// TIA Portal V16 export
// export: Created 2022-11-17T15:49:21.0130666Z, ExportSetting WithDefaults, DisplayName Totally Integrated Automation Portal, DisplayVersion V16 Update 6, DisplayName TIA Portal Version Control Interface, DisplayVersion V16 Update 2, DisplayName TIA Portal Openness, DisplayVersion V16 Update 6, DisplayName SINAMICS Startdrive Advanced, DisplayVersion V16 Update 5, DisplayName SINAMICS Startdrive G130, G150, S120, S150, SINAMICS MV, S210, DisplayVersion V16 Update 5, DisplayName SINAMICS Startdrive G110M, G120, G120C, G120D, G120P, G115D, DisplayVersion V16 Update 5, DisplayName STEP 7 Professional, DisplayVersion V16 Update 6, DisplayName STEP 7 Safety, DisplayVersion V16, DisplayName WinCC Advanced, DisplayVersion V16 Update 6
FUNCTION "FC27_PosSelfcEncoder" : Void   // FC27, LAD
TITLE = Pallet positioning with selfcentering system and encoder
{ S7_Optimized_Access := 'FALSE' }
AUTHOR : Robopac
VERSION : 0.0
// stored: AutoNumber false, IsIECCheckEnabled false, SetENOAutomatically false, UDAEnableTagReadback false
   VAR_TEMP
      Ch7ValmmEnco1 : DInt;
      Ch7ValmmEnco2 : DInt;
      PalletLenghtdiv2 : Int;
      PosToReach : Int;
      PosToDecelation : Int;
      WTemp1 : Int;
      DWTemp1 : DInt;
      DWTemp2 : DInt;
   END_VAR
   VAR_TEMP   // added for the SCL form of the ladder/FBD networks
      _w1 : Bool;
      _w2 : Bool;
   END_VAR
BEGIN

REGION Network 1: Delay on pallet positioning left
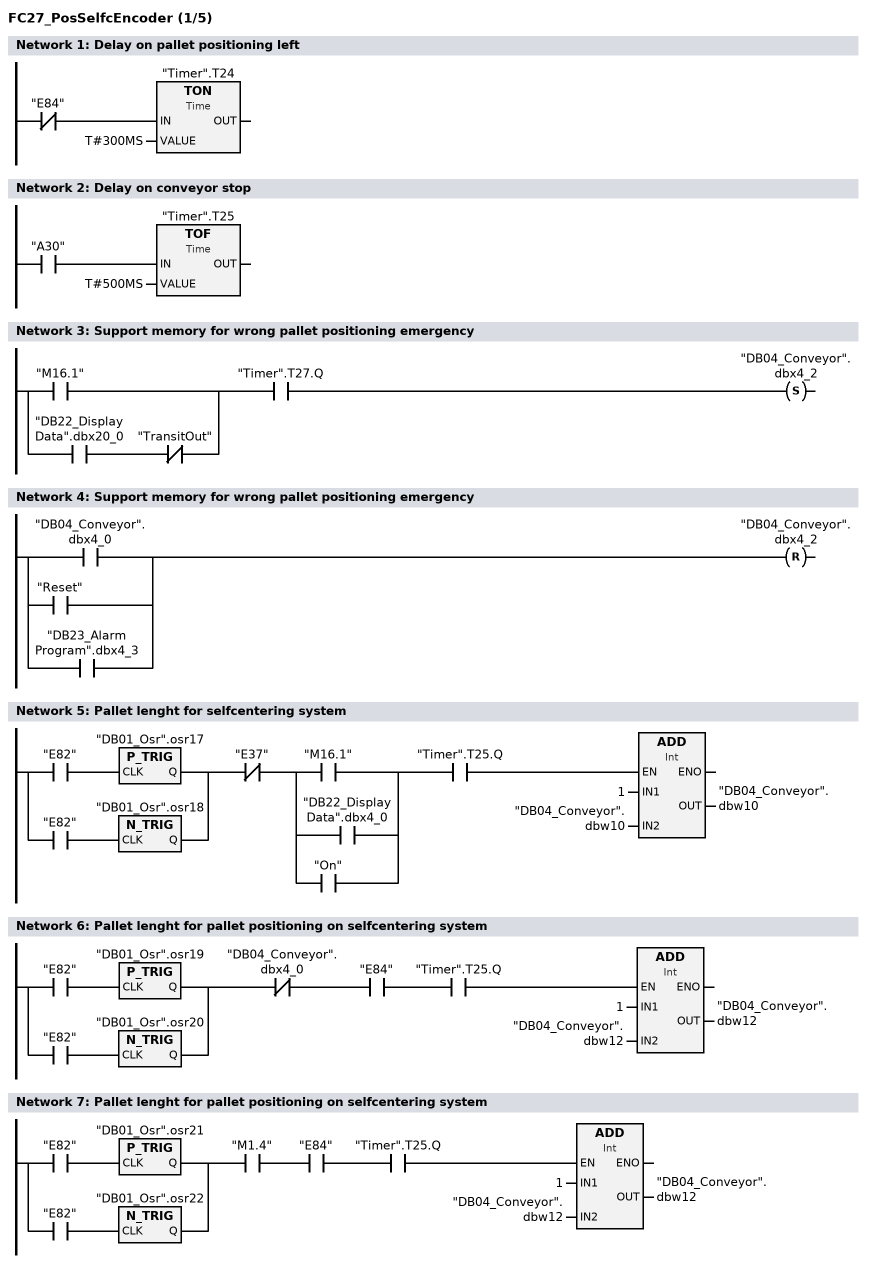
   "Timer".T24.TON(IN := NOT "E84", PT := T#300MS);   // TON coil
END_REGION

REGION Network 2: Delay on conveyor stop
   "Timer".T25.TOF(IN := "A30", PT := T#500MS);   // TOF coil
END_REGION

REGION Network 3: Support memory for wrong pallet positioning emergency
   RUNG wire#powerrail
      Contact( "M16.1" )
      wire#w1
      Contact( "Timer".T27.Q )
      S_Coil( "DB04_Conveyor".dbx4_2 )
   END_RUNG
   RUNG wire#powerrail
      Contact( "DB22_DisplayData".dbx20_0 )
      I_Contact( "TransitOut" )
   END_RUNG wire#w1
   // the same network as SCL:
   IF ("M16.1" OR ("DB22_DisplayData".dbx20_0 AND NOT "TransitOut")) AND "Timer".T27.Q THEN
       "DB04_Conveyor".dbx4_2 := TRUE;
   END_IF;
END_REGION

REGION Network 4: Support memory for wrong pallet positioning emergency
   RUNG wire#powerrail
      Contact( "DB04_Conveyor".dbx4_0 )
      wire#w1
      R_Coil( "DB04_Conveyor".dbx4_2 )
   END_RUNG
   RUNG wire#powerrail
      Contact( "Reset" )
   END_RUNG wire#w1
   RUNG wire#powerrail
      Contact( "DB23_AlarmProgram".dbx4_3 )
   END_RUNG wire#w1
   // the same network as SCL:
   IF "DB04_Conveyor".dbx4_0 OR "Reset" OR "DB23_AlarmProgram".dbx4_3 THEN
       "DB04_Conveyor".dbx4_2 := FALSE;
   END_IF;
END_REGION

REGION Network 5: Pallet lenght for selfcentering system
   RUNG wire#powerrail
      Contact( "E82" )
      P_Trig( "DB01_Osr".osr17 )
      wire#w1
      I_Contact( "E37" )
      wire#w2
      Contact( "M16.1" )
      wire#w3
      Contact( "Timer".T25.Q )
      { S7_Templates := "SrcType := Int"; S7_GenerateENO := "TRUE" } Add(in1 := 1, in2 := "DB04_Conveyor".dbw10, out => "DB04_Conveyor".dbw10)
   END_RUNG
   RUNG wire#powerrail
      Contact( "E82" )
      N_Trig( "DB01_Osr".osr18 )
   END_RUNG wire#w1
   RUNG wire#w2
      Contact( "DB22_DisplayData".dbx4_0 )
   END_RUNG wire#w3
   RUNG wire#w2
      Contact( "On" )
   END_RUNG wire#w3
   // the same network as SCL:
   #_w1 := "E82" AND NOT "DB01_Osr".osr17;   // rising edge
   "DB01_Osr".osr17 := "E82";
   #_w2 := NOT "E82" AND "DB01_Osr".osr18;   // falling edge
   "DB01_Osr".osr18 := "E82";
   IF (#_w1 OR #_w2) AND NOT "E37" AND ("M16.1" OR "DB22_DisplayData".dbx4_0 OR "On") AND "Timer".T25.Q THEN
       "DB04_Conveyor".dbw10 := 1 + "DB04_Conveyor".dbw10;
   END_IF;
END_REGION

REGION Network 6: Pallet lenght for pallet positioning on selfcentering system
   RUNG wire#powerrail
      Contact( "E82" )
      P_Trig( "DB01_Osr".osr19 )
      wire#w1
      I_Contact( "DB04_Conveyor".dbx4_0 )
      Contact( "E84" )
      Contact( "Timer".T25.Q )
      { S7_Templates := "SrcType := Int"; S7_GenerateENO := "TRUE" } Add(in1 := 1, in2 := "DB04_Conveyor".dbw12, out => "DB04_Conveyor".dbw12)
   END_RUNG
   RUNG wire#powerrail
      Contact( "E82" )
      N_Trig( "DB01_Osr".osr20 )
   END_RUNG wire#w1
   // the same network as SCL:
   #_w1 := "E82" AND NOT "DB01_Osr".osr19;   // rising edge
   "DB01_Osr".osr19 := "E82";
   #_w2 := NOT "E82" AND "DB01_Osr".osr20;   // falling edge
   "DB01_Osr".osr20 := "E82";
   IF (#_w1 OR #_w2) AND NOT "DB04_Conveyor".dbx4_0 AND "E84" AND "Timer".T25.Q THEN
       "DB04_Conveyor".dbw12 := 1 + "DB04_Conveyor".dbw12;
   END_IF;
END_REGION

REGION Network 7: Pallet lenght for pallet positioning on selfcentering system
   RUNG wire#powerrail
      Contact( "E82" )
      P_Trig( "DB01_Osr".osr21 )
      wire#w1
      Contact( "M1.4" )
      Contact( "E84" )
      Contact( "Timer".T25.Q )
      { S7_Templates := "SrcType := Int"; S7_GenerateENO := "TRUE" } Add(in1 := 1, in2 := "DB04_Conveyor".dbw12, out => "DB04_Conveyor".dbw12)
   END_RUNG
   RUNG wire#powerrail
      Contact( "E82" )
      N_Trig( "DB01_Osr".osr22 )
   END_RUNG wire#w1
   // the same network as SCL:
   #_w1 := "E82" AND NOT "DB01_Osr".osr21;   // rising edge
   "DB01_Osr".osr21 := "E82";
   #_w2 := NOT "E82" AND "DB01_Osr".osr22;   // falling edge
   "DB01_Osr".osr22 := "E82";
   IF (#_w1 OR #_w2) AND "M1.4" AND "E84" AND "Timer".T25.Q THEN
       "DB04_Conveyor".dbw12 := 1 + "DB04_Conveyor".dbw12;
   END_IF;
END_REGION

REGION Network 8: Reset pallet lenght
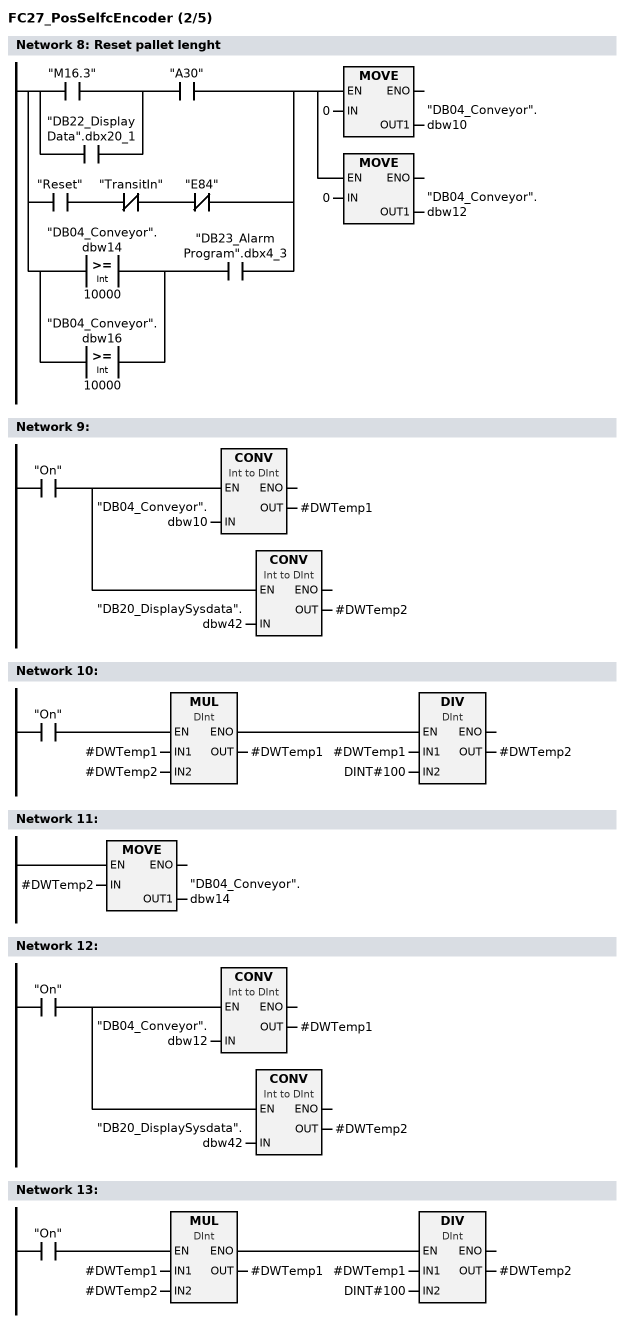
   RUNG wire#powerrail
      Contact( "M16.3" )
      wire#w1
      Contact( "A30" )
      wire#w2
      { S7_GenerateENO := "TRUE" } Move(in := 0, out1 => "DB04_Conveyor".dbw10)
   END_RUNG
   RUNG wire#powerrail
      Contact( "DB22_DisplayData".dbx20_1 )
   END_RUNG wire#w1
   RUNG wire#powerrail
      Contact( "Reset" )
      I_Contact( "TransitIn" )
      I_Contact( "E84" )
   END_RUNG wire#w2
   RUNG wire#powerrail
      { S7_Templates := "SrcType := Int" } GE_Contact(in1 := "DB04_Conveyor".dbw14, in2 := 10000)
      wire#w3
      Contact( "DB23_AlarmProgram".dbx4_3 )
   END_RUNG wire#w2
   RUNG wire#powerrail
      { S7_Templates := "SrcType := Int" } GE_Contact(in1 := "DB04_Conveyor".dbw16, in2 := 10000)
   END_RUNG wire#w3
   RUNG wire#w2
      { S7_GenerateENO := "TRUE" } Move(in := 0, out1 => "DB04_Conveyor".dbw12)
   END_RUNG
   // the same network as SCL:
   IF (("M16.3" OR "DB22_DisplayData".dbx20_1) AND "A30") OR ("Reset" AND NOT "TransitIn" AND NOT "E84") OR ((("DB04_Conveyor".dbw14 >= 10000) OR ("DB04_Conveyor".dbw16 >= 10000)) AND "DB23_AlarmProgram".dbx4_3) THEN
       "DB04_Conveyor".dbw10 := 0;
       "DB04_Conveyor".dbw12 := 0;
   END_IF;
END_REGION

REGION Network 9
   RUNG wire#powerrail
      Contact( "On" )
      wire#w1
      { S7_Templates := "[SrcType := Int, DestType := DInt]"; S7_GenerateENO := "TRUE" } Convert(in := "DB04_Conveyor".dbw10, out => #DWTemp1)
   END_RUNG
   RUNG wire#w1
      { S7_Templates := "[SrcType := Int, DestType := DInt]"; S7_GenerateENO := "TRUE" } Convert(in := "DB20_DisplaySysdata".dbw42, out => #DWTemp2)
   END_RUNG
   // the same network as SCL:
   IF "On" THEN
       #DWTemp1 := INT_TO_DINT("DB04_Conveyor".dbw10);
       #DWTemp2 := INT_TO_DINT("DB20_DisplaySysdata".dbw42);
   END_IF;
END_REGION

REGION Network 10
   RUNG wire#powerrail
      Contact( "On" )
      { S7_Templates := "SrcType := DInt"; S7_GenerateENO := "TRUE" } Mul(in1 := #DWTemp1, in2 := #DWTemp2, out => #DWTemp1)
      { S7_Templates := "SrcType := DInt"; S7_GenerateENO := "TRUE" } Div(in1 := #DWTemp1, in2 := DINT#100, out => #DWTemp2)
   END_RUNG
   // the same network as SCL:
   // ENO of a box is taken as its EN; it also drops when the box reports an error
   IF "On" THEN
       #DWTemp1 := #DWTemp1 * #DWTemp2;
       #DWTemp2 := #DWTemp1 / DINT#100;
   END_IF;
END_REGION

REGION Network 11
   RUNG wire#powerrail
      { S7_GenerateENO := "TRUE" } Move(in := #DWTemp2, out1 => "DB04_Conveyor".dbw14)
   END_RUNG
   // the same network as SCL:
   "DB04_Conveyor".dbw14 := #DWTemp2;
END_REGION

REGION Network 12
   RUNG wire#powerrail
      Contact( "On" )
      wire#w1
      { S7_Templates := "[SrcType := Int, DestType := DInt]"; S7_GenerateENO := "TRUE" } Convert(in := "DB04_Conveyor".dbw12, out => #DWTemp1)
   END_RUNG
   RUNG wire#w1
      { S7_Templates := "[SrcType := Int, DestType := DInt]"; S7_GenerateENO := "TRUE" } Convert(in := "DB20_DisplaySysdata".dbw42, out => #DWTemp2)
   END_RUNG
   // the same network as SCL:
   IF "On" THEN
       #DWTemp1 := INT_TO_DINT("DB04_Conveyor".dbw12);
       #DWTemp2 := INT_TO_DINT("DB20_DisplaySysdata".dbw42);
   END_IF;
END_REGION

REGION Network 13
   RUNG wire#powerrail
      Contact( "On" )
      { S7_Templates := "SrcType := DInt"; S7_GenerateENO := "TRUE" } Mul(in1 := #DWTemp1, in2 := #DWTemp2, out => #DWTemp1)
      { S7_Templates := "SrcType := DInt"; S7_GenerateENO := "TRUE" } Div(in1 := #DWTemp1, in2 := DINT#100, out => #DWTemp2)
   END_RUNG
   // the same network as SCL:
   // ENO of a box is taken as its EN; it also drops when the box reports an error
   IF "On" THEN
       #DWTemp1 := #DWTemp1 * #DWTemp2;
       #DWTemp2 := #DWTemp1 / DINT#100;
   END_IF;
END_REGION

REGION Network 14
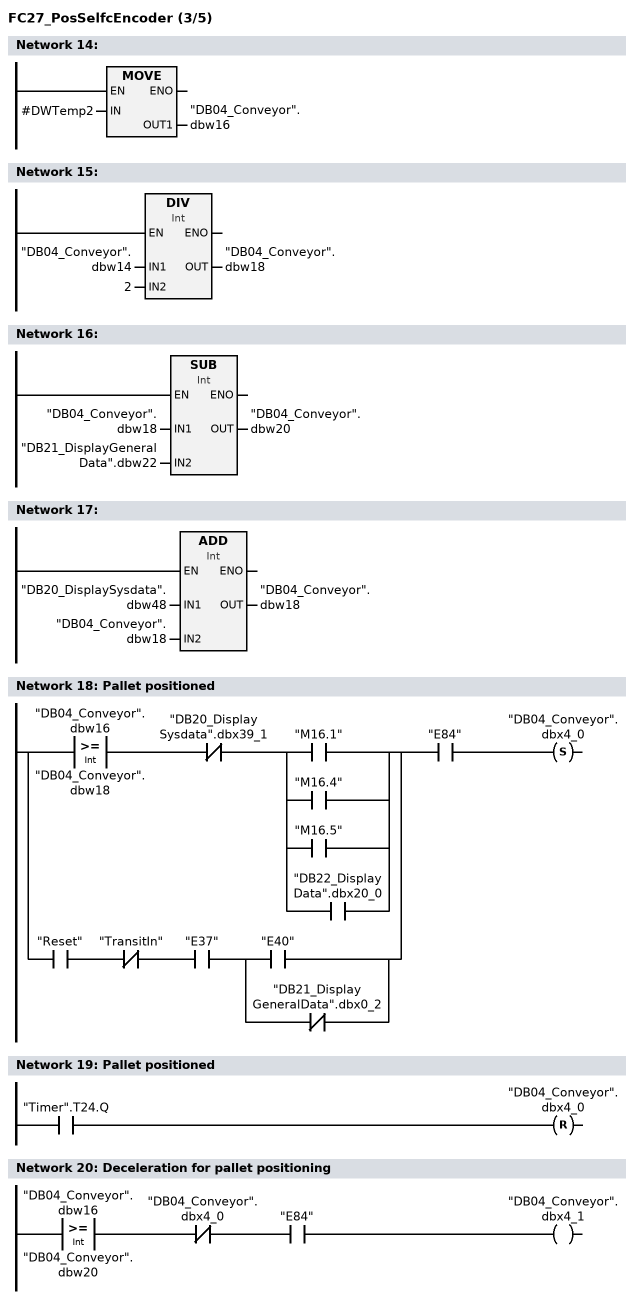
   RUNG wire#powerrail
      { S7_GenerateENO := "TRUE" } Move(in := #DWTemp2, out1 => "DB04_Conveyor".dbw16)
   END_RUNG
   // the same network as SCL:
   "DB04_Conveyor".dbw16 := #DWTemp2;
END_REGION

REGION Network 15
   RUNG wire#powerrail
      { S7_Templates := "SrcType := Int"; S7_GenerateENO := "TRUE" } Div(in1 := "DB04_Conveyor".dbw14, in2 := 2, out => "DB04_Conveyor".dbw18)
   END_RUNG
   // the same network as SCL:
   "DB04_Conveyor".dbw18 := "DB04_Conveyor".dbw14 / 2;
END_REGION

REGION Network 16
   RUNG wire#powerrail
      { S7_Templates := "SrcType := Int"; S7_GenerateENO := "TRUE" } Sub(in1 := "DB04_Conveyor".dbw18, in2 := "DB21_DisplayGeneralData".dbw22, out => "DB04_Conveyor".dbw20)
   END_RUNG
   // the same network as SCL:
   "DB04_Conveyor".dbw20 := "DB04_Conveyor".dbw18 - "DB21_DisplayGeneralData".dbw22;
END_REGION

REGION Network 17
   RUNG wire#powerrail
      { S7_Templates := "SrcType := Int"; S7_GenerateENO := "TRUE" } Add(in1 := "DB20_DisplaySysdata".dbw48, in2 := "DB04_Conveyor".dbw18, out => "DB04_Conveyor".dbw18)
   END_RUNG
   // the same network as SCL:
   "DB04_Conveyor".dbw18 := "DB20_DisplaySysdata".dbw48 + "DB04_Conveyor".dbw18;
END_REGION

REGION Network 18: Pallet positioned
   RUNG wire#powerrail
      { S7_Templates := "SrcType := Int" } GE_Contact(in1 := "DB04_Conveyor".dbw16, in2 := "DB04_Conveyor".dbw18)
      I_Contact( "DB20_DisplaySysdata".dbx39_1 )
      wire#w1
      Contact( "M16.1" )
      wire#w2
      Contact( "E84" )
      S_Coil( "DB04_Conveyor".dbx4_0 )
   END_RUNG
   RUNG wire#w1
      Contact( "M16.4" )
   END_RUNG wire#w2
   RUNG wire#w1
      Contact( "M16.5" )
   END_RUNG wire#w2
   RUNG wire#w1
      Contact( "DB22_DisplayData".dbx20_0 )
   END_RUNG wire#w2
   RUNG wire#powerrail
      Contact( "Reset" )
      I_Contact( "TransitIn" )
      Contact( "E37" )
      wire#w3
      Contact( "E40" )
   END_RUNG wire#w2
   RUNG wire#w3
      I_Contact( "DB21_DisplayGeneralData".dbx0_2 )
   END_RUNG wire#w2
   // the same network as SCL:
   IF ((("DB04_Conveyor".dbw16 >= "DB04_Conveyor".dbw18) AND NOT "DB20_DisplaySysdata".dbx39_1 AND ("M16.1" OR "M16.4" OR "M16.5" OR "DB22_DisplayData".dbx20_0)) OR ("Reset" AND NOT "TransitIn" AND "E37" AND ("E40" OR NOT "DB21_DisplayGeneralData".dbx0_2))) AND "E84" THEN
       "DB04_Conveyor".dbx4_0 := TRUE;
   END_IF;
END_REGION

REGION Network 19: Pallet positioned
   RUNG wire#powerrail
      Contact( "Timer".T24.Q )
      R_Coil( "DB04_Conveyor".dbx4_0 )
   END_RUNG
   // the same network as SCL:
   IF "Timer".T24.Q THEN "DB04_Conveyor".dbx4_0 := FALSE; END_IF;
END_REGION

REGION Network 20: Deceleration for pallet positioning
   RUNG wire#powerrail
      { S7_Templates := "SrcType := Int" } GE_Contact(in1 := "DB04_Conveyor".dbw16, in2 := "DB04_Conveyor".dbw20)
      I_Contact( "DB04_Conveyor".dbx4_0 )
      Contact( "E84" )
      Coil( "DB04_Conveyor".dbx4_1 )
   END_RUNG
   // the same network as SCL:
   "DB04_Conveyor".dbx4_1 := ("DB04_Conveyor".dbw16 >= "DB04_Conveyor".dbw20) AND NOT "DB04_Conveyor".dbx4_0 AND "E84";
END_REGION

REGION Network 21: Short pallet positioned
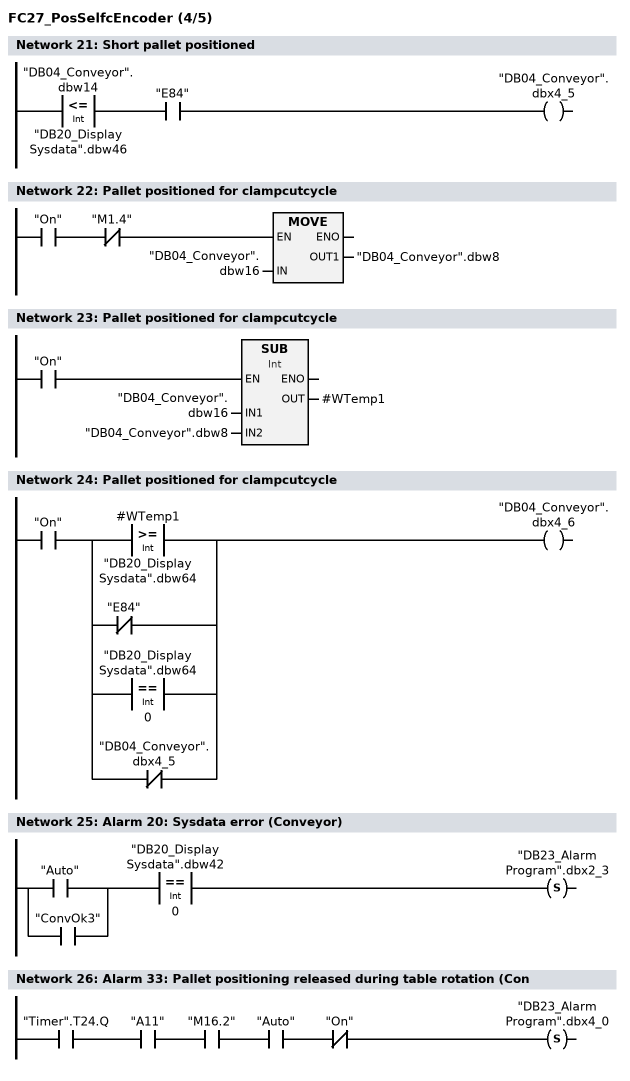
   RUNG wire#powerrail
      { S7_Templates := "SrcType := Int" } LE_Contact(in1 := "DB04_Conveyor".dbw14, in2 := "DB20_DisplaySysdata".dbw46)
      Contact( "E84" )
      Coil( "DB04_Conveyor".dbx4_5 )
   END_RUNG
   // the same network as SCL:
   "DB04_Conveyor".dbx4_5 := ("DB04_Conveyor".dbw14 <= "DB20_DisplaySysdata".dbw46) AND "E84";
END_REGION

REGION Network 22: Pallet positioned for clampcutcycle
   RUNG wire#powerrail
      Contact( "On" )
      I_Contact( "M1.4" )
      { S7_GenerateENO := "TRUE" } Move(in := "DB04_Conveyor".dbw16, out1 => "DB04_Conveyor".dbw8)
   END_RUNG
   // the same network as SCL:
   IF "On" AND NOT "M1.4" THEN "DB04_Conveyor".dbw8 := "DB04_Conveyor".dbw16; END_IF;
END_REGION

REGION Network 23: Pallet positioned for clampcutcycle
   RUNG wire#powerrail
      Contact( "On" )
      { S7_Templates := "SrcType := Int"; S7_GenerateENO := "TRUE" } Sub(in1 := "DB04_Conveyor".dbw16, in2 := "DB04_Conveyor".dbw8, out => #WTemp1)
   END_RUNG
   // the same network as SCL:
   IF "On" THEN #WTemp1 := "DB04_Conveyor".dbw16 - "DB04_Conveyor".dbw8; END_IF;
END_REGION

REGION Network 24: Pallet positioned for clampcutcycle
   RUNG wire#powerrail
      Contact( "On" )
      wire#w1
      { S7_Templates := "SrcType := Int" } GE_Contact(in1 := #WTemp1, in2 := "DB20_DisplaySysdata".dbw64)
      wire#w2
      Coil( "DB04_Conveyor".dbx4_6 )
   END_RUNG
   RUNG wire#w1
      I_Contact( "E84" )
   END_RUNG wire#w2
   RUNG wire#w1
      { S7_Templates := "SrcType := Int" } EQ_Contact(in1 := "DB20_DisplaySysdata".dbw64, in2 := 0)
   END_RUNG wire#w2
   RUNG wire#w1
      I_Contact( "DB04_Conveyor".dbx4_5 )
   END_RUNG wire#w2
   // the same network as SCL:
   "DB04_Conveyor".dbx4_6 := "On" AND ((#WTemp1 >= "DB20_DisplaySysdata".dbw64) OR NOT "E84" OR ("DB20_DisplaySysdata".dbw64 = 0) OR NOT "DB04_Conveyor".dbx4_5);
END_REGION

REGION Network 25: Alarm 20: Sysdata error (Conveyor)
   RUNG wire#powerrail
      Contact( "Auto" )
      wire#w1
      { S7_Templates := "SrcType := Int" } EQ_Contact(in1 := "DB20_DisplaySysdata".dbw42, in2 := 0)
      S_Coil( "DB23_AlarmProgram".dbx2_3 )
   END_RUNG
   RUNG wire#powerrail
      Contact( "ConvOk3" )
   END_RUNG wire#w1
   // the same network as SCL:
   IF ("Auto" OR "ConvOk3") AND ("DB20_DisplaySysdata".dbw42 = 0) THEN
       "DB23_AlarmProgram".dbx2_3 := TRUE;
   END_IF;
END_REGION

REGION Network 26: Alarm 33: Pallet positioning released during table rotation (Con
   RUNG wire#powerrail
      Contact( "Timer".T24.Q )
      Contact( "A11" )
      Contact( "M16.2" )
      Contact( "Auto" )
      I_Contact( "On" )
      S_Coil( "DB23_AlarmProgram".dbx4_0 )
   END_RUNG
   // the same network as SCL:
   IF "Timer".T24.Q AND "A11" AND "M16.2" AND "Auto" AND NOT "On" THEN
       "DB23_AlarmProgram".dbx4_0 := TRUE;
   END_IF;
END_REGION

REGION Network 27: Alarm 36: Wrong pallet positioning (Conveyor)
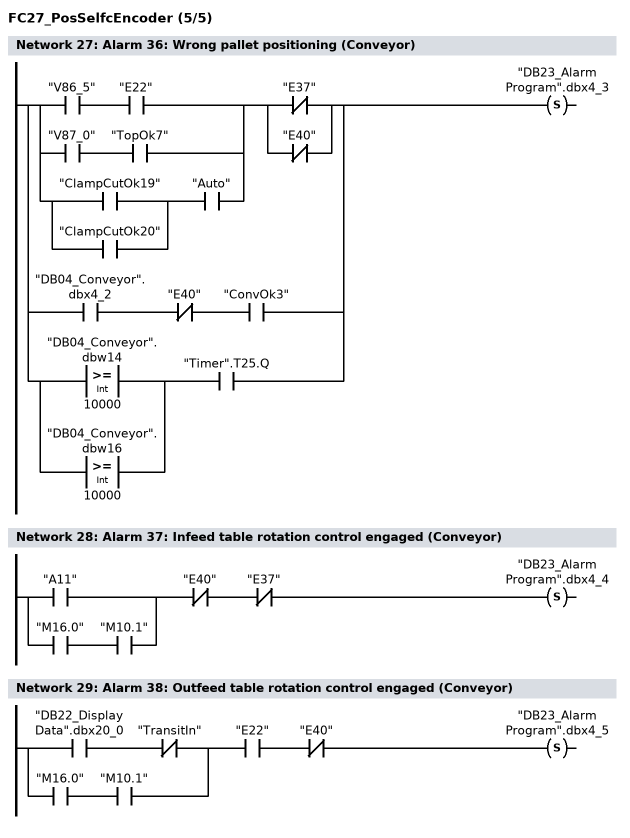
   RUNG wire#powerrail
      Contact( "V86_5" )
      Contact( "E22" )
      wire#w1
      I_Contact( "E37" )
      wire#w3
      S_Coil( "DB23_AlarmProgram".dbx4_3 )
   END_RUNG
   RUNG wire#powerrail
      Contact( "V87_0" )
      Contact( "TopOk7" )
   END_RUNG wire#w1
   RUNG wire#powerrail
      Contact( "ClampCutOk19" )
      wire#w2
      Contact( "Auto" )
   END_RUNG wire#w1
   RUNG wire#powerrail
      Contact( "ClampCutOk20" )
   END_RUNG wire#w2
   RUNG wire#w1
      I_Contact( "E40" )
   END_RUNG wire#w3
   RUNG wire#powerrail
      Contact( "DB04_Conveyor".dbx4_2 )
      I_Contact( "E40" )
      Contact( "ConvOk3" )
   END_RUNG wire#w3
   RUNG wire#powerrail
      { S7_Templates := "SrcType := Int" } GE_Contact(in1 := "DB04_Conveyor".dbw14, in2 := 10000)
      wire#w4
      Contact( "Timer".T25.Q )
   END_RUNG wire#w3
   RUNG wire#powerrail
      { S7_Templates := "SrcType := Int" } GE_Contact(in1 := "DB04_Conveyor".dbw16, in2 := 10000)
   END_RUNG wire#w4
   // the same network as SCL:
   IF ((("V86_5" AND "E22") OR ("V87_0" AND "TopOk7") OR (("ClampCutOk19" OR "ClampCutOk20") AND "Auto")) AND (NOT "E37" OR NOT "E40")) OR ("DB04_Conveyor".dbx4_2 AND NOT "E40" AND "ConvOk3") OR ((("DB04_Conveyor".dbw14 >= 10000) OR ("DB04_Conveyor".dbw16 >= 10000)) AND "Timer".T25.Q) THEN
       "DB23_AlarmProgram".dbx4_3 := TRUE;
   END_IF;
END_REGION

REGION Network 28: Alarm 37: Infeed table rotation control engaged (Conveyor)
   RUNG wire#powerrail
      Contact( "A11" )
      wire#w1
      I_Contact( "E40" )
      I_Contact( "E37" )
      S_Coil( "DB23_AlarmProgram".dbx4_4 )
   END_RUNG
   RUNG wire#powerrail
      Contact( "M16.0" )
      Contact( "M10.1" )
   END_RUNG wire#w1
   // the same network as SCL:
   IF ("A11" OR ("M16.0" AND "M10.1")) AND NOT "E40" AND NOT "E37" THEN
       "DB23_AlarmProgram".dbx4_4 := TRUE;
   END_IF;
END_REGION

REGION Network 29: Alarm 38: Outfeed table rotation control engaged (Conveyor)
   RUNG wire#powerrail
      Contact( "DB22_DisplayData".dbx20_0 )
      I_Contact( "TransitIn" )
      wire#w1
      Contact( "E22" )
      I_Contact( "E40" )
      S_Coil( "DB23_AlarmProgram".dbx4_5 )
   END_RUNG
   RUNG wire#powerrail
      Contact( "M16.0" )
      Contact( "M10.1" )
   END_RUNG wire#w1
   // the same network as SCL:
   IF (("DB22_DisplayData".dbx20_0 AND NOT "TransitIn") OR ("M16.0" AND "M10.1")) AND "E22" AND NOT "E40" THEN
       "DB23_AlarmProgram".dbx4_5 := TRUE;
   END_IF;
END_REGION
END_FUNCTION
